INTERFACE I_InstanceAddedEvent EXTENDS I_Event

PROPERTY PUBLIC Instance : I_Instance
GET
END_GET
END_PROPERTY

END_INTERFACE

(* stored: Version 1.1.0.1, ProductVersion 3.1.4024.11
   Itf I_InstanceAddedEvent: Id {3198bc2b-c515-452e-b40b-7d74c05c9b69}
   Property Instance: Id {17d0bbfd-e826-4602-b939-ce91fc65d8a7}
   Get Get: Id {f8f90cc4-4659-47cd-8f63-f0a93e5d499d} *)
